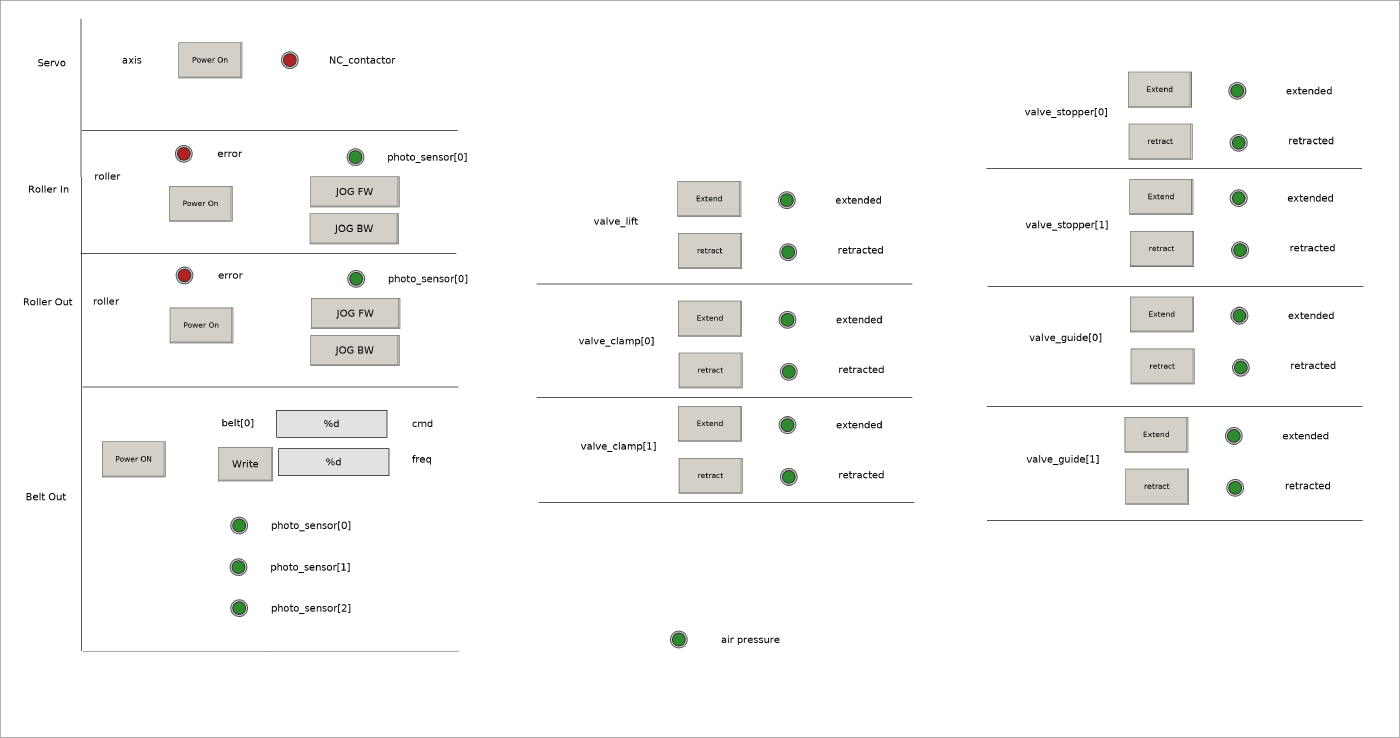
VISUALIZATION v_IO_LC  // 2048x1080
VAR_IN_OUT
	dIO_LC		: LateralRecy_Module;
END_VAR
    Lamp1 (505,215 30x30), variable: dIO_LC.rollerIn.photo_sensor, style: Lamp-Lamp1-Green
    Label (559,217 132x26), "photo_sensor[0]"
    Label (31,264 80x26), "Roller In"
    Lamp1 (254,210 30x30), variable: dIO_LC.rollerIn.roller.err, style: Lamp-Lamp1-Red
    Label (270,212 132x26), "error"
    Label (91,245 132x26), "roller"
    Line (120,190) (669,190)
    Line (118,28) (119,952)
    Button (454,258 130x45), "JOG FW", colour toggle: dIO_LC.rollerIn.roller.forward
        OnMouseDown: execute { dIO_LC.rollerIn.roller.forward := TRUE; }
        OnMouseUp: execute { dIO_LC.rollerIn.roller.forward := FALSE; }
    Button (453,312 130x45), "JOG BW", colour toggle: dIO_LC.rollerIn.roller.backward
        OnMouseDown: execute { dIO_LC.rollerIn.roller.backward := TRUE; }
        OnMouseUp: execute { dIO_LC.rollerIn.roller.backward := FALSE; }
    Button (247,272 93x52), "Power On", colour toggle: dIO_LC.rollerIn.roller.Power
        toggle dIO_LC.rollerIn.roller.Power
    Line (118,370) (667,370)
    Line (121,566) (670,566)
    Label (1480,151 160x26), "valve_stopper[0]"
    Button (1650,105 93x52), "Extend", colour toggle: dIO_LC.valve_stopper[0].extend
        OnMouseDown: execute { dIO_LC.valve_stopper[0].extend := TRUE; dIO_LC.valve_stopper[0].retract := FALSE; }
    Button (1651,181 93x52), "retract", colour toggle: dIO_LC.valve_stopper[0].retract
        OnMouseDown: execute { dIO_LC.valve_stopper[0].extend := FALSE; dIO_LC.valve_stopper[0].retract := TRUE; }
    Lamp1 (1795,118 30x30), variable: dIO_LC.valve_stopper[0].extended, style: Lamp-Lamp1-Green
    Lamp1 (1797,194 30x30), variable: dIO_LC.valve_stopper[0].retracted, style: Lamp-Lamp1-Green
    Label (1849,120 132x26), "extended"
    Label (1852,193 132x26), "retracted"
    Label (1481,316 160x26), "valve_stopper[1]"
    Label (1479,481 160x26), "valve_guide[0]"
    Label (1475,659 160x26), "valve_guide[1]"
    Line (1443,246) (1992,246)
    Line (1445,419) (1994,419)
    Line (1444,594) (1993,594)
    Line (1444,761) (1993,761)
    Label (89,428 132x26), "roller"
    Label (30,429 80x26), "Roller Out"
    Rectangle (404,600 162x40), "%d", text variable: dIO_LC.belt_out.belt.fbconverter.cmd
        OnMouseClick: write the text variable via Default
    Rectangle (407,656 162x40), "%d", text variable: dIO_LC.belt_out.belt.fbconverter.freq
        OnMouseClick: write the text variable via Default
    Label (282,606 132x26), "belt[0]"
    Label (552,607 132x26), "cmd"
    Label (551,659 132x26), "freq"
    Button (149,646 93x52), "Power ON", colour toggle: dIO_LC.power_beltConv
        toggle dIO_LC.power_beltConv
    Button (319,654 80x50), "Write"
        OnMouseDown: execute { dIO_LC.belt_out.belt.fbconverter.bSetParaEx	:= TRUE; }
        OnMouseUp: execute { dIO_LC.belt_out.belt.fbconverter.bSetParaEx	:= FALSE; }
    Lamp1 (335,754 30x30), variable: dIO_LC.belt_out.photo_sensor[0], style: Lamp-Lamp1-Green
    Label (389,756 132x26), "photo_sensor[0]"
    Lamp1 (334,815 30x30), variable: dIO_LC.belt_out.photo_sensor[1], style: Lamp-Lamp1-Green
    Label (388,817 132x26), "photo_sensor[1]"
    Lamp1 (335,875 30x30), variable: dIO_LC.belt_out.photo_sensor[2], style: Lamp-Lamp1-Green
    Label (389,877 132x26), "photo_sensor[2]"
    Label (464,75 132x26), "NC_contactor"
    Label (127,75 132x26), "axis"
    Button (261,62 93x52), "Power On", colour toggle: dIO_LC.lateral.power_axis
        toggle dIO_LC.lateral.power_axis
    Lamp1 (409,73 30x30), variable: dIO_LC.lateral.contactor_axis, style: Lamp-Lamp1-Red
    Label (821,311 160x26), "valve_lift"
    Button (991,265 93x52), "Extend", colour toggle: dIO_LC.lateral.valve_lift.extend
        OnMouseDown: execute { dIO_LC.lateral.valve_lift.extend := TRUE; dIO_LC.lateral.valve_lift.retract := FALSE; }
    Button (992,341 93x52), "retract", colour toggle: dIO_LC.lateral.valve_lift.retract
        OnMouseDown: execute { dIO_LC.lateral.valve_lift.extend := FALSE; dIO_LC.lateral.valve_lift.retract := TRUE; }
    Lamp1 (1136,278 30x30), variable: dIO_LC.lateral.valve_lift.extended, style: Lamp-Lamp1-Green
    Lamp1 (1138,354 30x30), variable: dIO_LC.lateral.valve_lift.retracted, style: Lamp-Lamp1-Green
    Label (1190,280 132x26), "extended"
    Label (1193,353 132x26), "retracted"
    Label (822,486 160x26), "valve_clamp[0]"
    Button (992,440 93x52), "Extend", colour toggle: dIO_LC.lateral.valve_clamp[0].extend
        OnMouseDown: execute { dIO_LC.lateral.valve_clamp[0].extend := TRUE; dIO_LC.lateral.valve_clamp[0].retract := FALSE; }
    Button (993,516 93x52), "retract", colour toggle: dIO_LC.lateral.valve_clamp[0].retract
        OnMouseDown: execute { dIO_LC.lateral.valve_clamp[0].extend := FALSE; dIO_LC.lateral.valve_clamp[0].retract := TRUE; }
    Lamp1 (1137,453 30x30), variable: dIO_LC.lateral.valve_clamp[0].extended, style: Lamp-Lamp1-Green
    Lamp1 (1139,529 30x30), variable: dIO_LC.lateral.valve_clamp[0].retracted, style: Lamp-Lamp1-Green
    Label (1191,455 132x26), "extended"
    Label (1194,528 132x26), "retracted"
    Line (785,581) (1334,581)
    Label (825,640 160x26), "valve_clamp[1]"
    Line (788,735) (1337,735)
    Line (785,415) (1334,415)
    Line (122,953) (671,952)
    Label (27,714 80x26), "Belt Out"
    Label (36,79 80x26), "Servo"
    Lamp1 (506,393 30x30), variable: dIO_LC.rollerOut.photo_sensor, style: Lamp-Lamp1-Green
    Label (560,395 132x26), "photo_sensor[0]"
    Lamp1 (255,388 30x30), variable: dIO_LC.rollerOut.roller.err, style: Lamp-Lamp1-Red
    Label (271,390 132x26), "error"
    Button (455,436 130x45), "JOG FW", colour toggle: dIO_LC.rollerOut.roller.forward
        OnMouseDown: execute { dIO_LC.rollerOut.roller.forward := TRUE; }
        OnMouseUp: execute { dIO_LC.rollerOut.roller.forward := FALSE; }
    Button (454,490 130x45), "JOG BW", colour toggle: dIO_LC.rollerOut.roller.backward
        OnMouseDown: execute { dIO_LC.rollerOut.roller.backward := TRUE; }
        OnMouseUp: execute { dIO_LC.rollerOut.roller.backward := FALSE; }
    Button (248,450 93x52), "Power On", colour toggle: dIO_LC.rollerOut.roller.Power
        toggle dIO_LC.rollerOut.roller.Power
    Button (992,594 93x52), "Extend", colour toggle: dIO_LC.lateral.valve_clamp[1].extend
        OnMouseDown: execute { dIO_LC.lateral.valve_clamp[1].extend := TRUE; dIO_LC.lateral.valve_clamp[1].retract := FALSE; }
    Button (993,670 93x52), "retract", colour toggle: dIO_LC.lateral.valve_clamp[1].retract
        OnMouseDown: execute { dIO_LC.lateral.valve_clamp[1].extend := FALSE; dIO_LC.lateral.valve_clamp[1].retract := TRUE; }
    Lamp1 (1137,607 30x30), variable: dIO_LC.lateral.valve_clamp[1].extended, style: Lamp-Lamp1-Green
    Lamp1 (1139,683 30x30), variable: dIO_LC.lateral.valve_clamp[1].retracted, style: Lamp-Lamp1-Green
    Label (1191,609 132x26), "extended"
    Label (1194,682 132x26), "retracted"
    Button (1652,262 93x52), "Extend", colour toggle: dIO_LC.valve_stopper[1].extend
        OnMouseDown: execute { dIO_LC.valve_stopper[1].extend := TRUE; dIO_LC.valve_stopper[1].retract := FALSE; }
    Button (1653,338 93x52), "retract", colour toggle: dIO_LC.valve_stopper[1].retract
        OnMouseDown: execute { dIO_LC.valve_stopper[1].extend := FALSE; dIO_LC.valve_stopper[1].retract := TRUE; }
    Lamp1 (1797,275 30x30), variable: dIO_LC.valve_stopper[1].extended, style: Lamp-Lamp1-Green
    Lamp1 (1799,351 30x30), variable: dIO_LC.valve_stopper[1].retracted, style: Lamp-Lamp1-Green
    Label (1851,277 132x26), "extended"
    Label (1854,350 132x26), "retracted"
    Button (1653,434 93x52), "Extend", colour toggle: dIO_LC.valve_guide[0].extend
        OnMouseDown: execute { dIO_LC.valve_guide[0].extend := TRUE; dIO_LC.valve_guide[0].retract := FALSE; }
    Button (1654,510 93x52), "retract", colour toggle: dIO_LC.valve_guide[0].retract
        OnMouseDown: execute { dIO_LC.valve_guide[0].extend := FALSE; dIO_LC.valve_guide[0].retract := TRUE; }
    Lamp1 (1798,447 30x30), variable: dIO_LC.valve_guide[0].extended, style: Lamp-Lamp1-Green
    Lamp1 (1800,523 30x30), variable: dIO_LC.valve_guide[0].retracted, style: Lamp-Lamp1-Green
    Label (1852,449 132x26), "extended"
    Label (1855,522 132x26), "retracted"
    Button (1645,610 93x52), "Extend", colour toggle: dIO_LC.valve_guide[1].extend
        OnMouseDown: execute { dIO_LC.valve_guide[1].extend := TRUE; dIO_LC.valve_guide[1].retract := FALSE; }
    Button (1646,686 93x52), "retract", colour toggle: dIO_LC.valve_guide[1].retract
        OnMouseDown: execute { dIO_LC.valve_guide[1].extend := FALSE; dIO_LC.valve_guide[1].retract := TRUE; }
    Lamp1 (1790,623 30x30), variable: dIO_LC.valve_guide[1].extended, style: Lamp-Lamp1-Green
    Lamp1 (1792,699 30x30), variable: dIO_LC.valve_guide[1].retracted, style: Lamp-Lamp1-Green
    Label (1844,625 132x26), "extended"
    Label (1847,698 132x26), "retracted"
    Lamp1 (978,921 30x30), variable: dIO_LC.pressure_sensor, style: Lamp-Lamp1-Green
    Label (1032,923 132x26), "air pressure"
END_VISUALIZATION

(* stored: Version 1.1.0.1, ProductVersion 3.1.4024.12
   Visu v_IO_LC: Id {1b271db9-cf41-41c9-9c7f-ea230d750d8a} *)
